INTERFACE I_Skill_Roboter_Erweitert

METHOD M_Reset : BOOL
VAR_INPUT
END_VAR
END_METHOD

METHOD M_Start : BOOL
VAR_INPUT
END_VAR
END_METHOD

METHOD M_Stop : BOOL
VAR_INPUT
END_VAR
END_METHOD

PROPERTY P_Erreicht : sKraftVariablen
SET
END_SET
END_PROPERTY

PROPERTY P_Limit : sKraftVariablen
SET
END_SET
END_PROPERTY

PROPERTY P_Roboterposition : sRoboterProzessVariablen
SET
END_SET
END_PROPERTY

PROPERTY P_State : eSkillState
GET
END_GET
END_PROPERTY

END_INTERFACE

(* stored: Version 1.1.0.1
   Itf I_Skill_Roboter_Erweitert: Id {56be7f36-2ba2-4a62-ac0c-da988620b2cd}
   Method M_Reset: Id {d3fa8aad-0eba-4efe-a62e-622566017fb9}
   Method M_Start: Id {f996823d-0a6a-4b75-a29d-925b0e03a6fd}
   Method M_Stop: Id {b503c177-c0b8-4e3f-b975-9d18dcfc89ee}
   Property P_Erreicht: Id {6401b69d-71a1-4968-9df2-e69ab692064e}
   Set Set: Id {738ada45-7ba2-4158-9703-1cc297d505a6}
   Property P_Limit: Id {2fa88caf-d84b-4b2b-8259-00c40bd917fe}
   Set Set: Id {fd81d98f-d438-403f-9d2d-5c6b7caede69}
   Property P_Roboterposition: Id {f0d7b625-f54b-4284-9533-fc10bd07b59e}
   Set Set: Id {1b10dff8-a1dc-410f-8fe5-b6b5271371f4}
   Property P_State: Id {b402ea62-4909-47be-bc64-47bdef77291f}
   Get Get: Id {77fec5d9-b2da-49ee-9fb6-a5ff3f3fada2} *)
